FUNCTION_BLOCK MoveValve (* Basic Function Block Type *)
  (* Standard: 61499-2 *)
  (* Version 0.0, 5/27/2016, Andrei, nxtControl GmbH, Template *)
  PACKAGE Main;
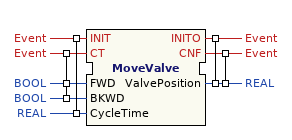
  EVENT_INPUT
    INIT WITH CycleTime; (* Initialization Request *)
    CT WITH FWD, BKWD;
  END_EVENT
  EVENT_OUTPUT
    INITO WITH ValvePosition; (* Initialization Confirm *)
    CNF WITH ValvePosition; (* Execution Confirmation *)
  END_EVENT
  VAR_INPUT
    FWD : BOOL; (* Input event qualifier *)
    BKWD : BOOL;
    CycleTime : REAL;
  END_VAR
  VAR_OUTPUT
    ValvePosition : REAL; (* Output event qualifier *)
  END_VAR
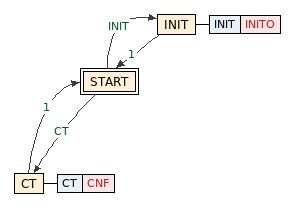
  EC_STATES
    START; (* Initial State *)
    INIT : INIT -> INITO; (* Initialization *)
    CT : CT -> CNF; (* Normal execution *)
  END_STATES
  EC_TRANSITIONS
    START TO INIT := INIT;
    INIT TO START := 1;
    START TO CT := CT;
    CT TO START := 1;
  END_TRANSITIONS
  ALGORITHM INIT IN ST: (* Initialization algorithm *)
ValvePosition := 0.0;
  END_ALGORITHM
  ALGORITHM CT IN ST: (* Normally executed algorithm *)
IF FWD AND NOT(BKWD) AND (ValvePosition + 200*CycleTime < 43.0) THEN
	ValvePosition := ValvePosition + 200*CycleTime;
ELSIF FWD AND NOT(BKWD) AND (ValvePosition + 200*CycleTime > 43.0) THEN
	ValvePosition := 43.0;
ELSIF NOT(FWD) AND BKWD AND (ValvePosition - 200*CycleTime > 0.0) THEN
	ValvePosition := ValvePosition - 200*CycleTime;
ELSIF NOT(FWD) AND BKWD AND (ValvePosition - 200*CycleTime < 0.0) THEN
	ValvePosition := 0.0;
ELSIF NOT(FWD) AND NOT(BKWD) THEN
	ValvePosition := -1.0;
ELSE
	ValvePosition := ValvePosition;
END_IF;
  END_ALGORITHM
END_FUNCTION_BLOCK
